// LS Electric XG5000 project: 66_3_A
// PLC NewPLC
// module base 0 slot 0: 입출력 모듈:XBC-DR20S (DC 24V 입력 12점, 릴레이 출력 8점)

PROGRAM NewProgram (task: 스캔 프로그램)

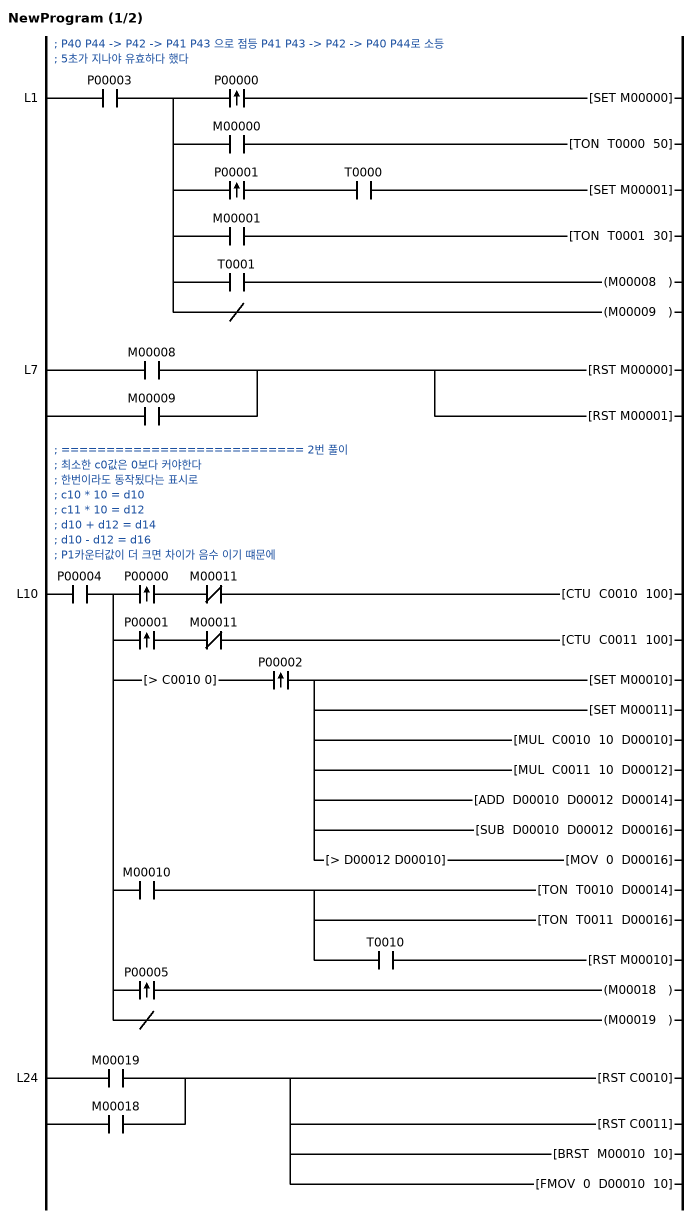
// P40 P44 -> P42 -> P41 P43 으로 점등 P41 P43 -> P42 -> P40 P44로 소등
; L1
LOAD      P00003
MPUSH
ANDP      P00000
SET       M00000
MLOAD
AND       M00000
TON       T0000 50
MLOAD
ANDP      P00001
AND       T0000
SET       M00001
MLOAD
AND       M00001
TON       T0001 30
MLOAD
AND       T0001
OUT       M00008
MPOP
NOT
OUT       M00009
// output comment: 5초가 지나야 유효하다 했다
; L7
LOAD      M00008
OR        M00009
RST       M00000
RST       M00001
// =========================== 2번 풀이
; L10
LOAD      P00004
MPUSH
ANDP      P00000
AND NOT   M00011
CTU       C0010 100
MLOAD
ANDP      P00001
AND NOT   M00011
CTU       C0011 100
MLOAD
AND>      C0010 0
ANDP      P00002
SET       M00010
SET       M00011
MUL       C0010 10 D00010
MUL       C0011 10 D00012
ADD       D00010 D00012 D00014
SUB       D00010 D00012 D00016
AND>      D00012 D00010
MOV       0 D00016
MLOAD
AND       M00010
TON       T0010 D00014
TON       T0011 D00016
AND       T0010
RST       M00010
MLOAD
ANDP      P00005
OUT       M00018
MPOP
NOT
OUT       M00019
// output comment: 
// output comment: 최소한 c0값은 0보다 커야한다
// output comment: 한번이라도 동작됬다는 표시로
// output comment: c10 * 10 = d10
// output comment: c11 * 10 = d12
// output comment: d10 + d12 = d14
// output comment: d10 - d12 = d16
// output comment: P1카운터값이 더 크면 차이가 음수 이기 떄문에
; L24
LOAD      M00019
OR        M00018
RST       C0010
RST       C0011
BRST      M00010 10
FMOV      0 D00010 10

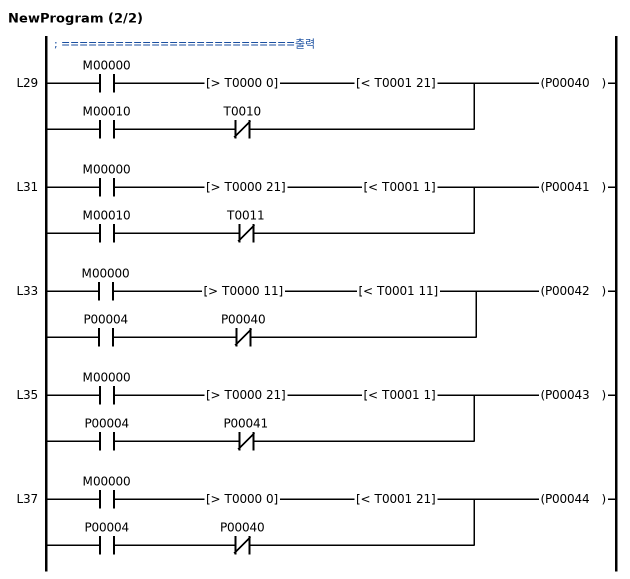
// ==========================출력
; L29
LOAD      M00000
AND>      T0000 0
AND<      T0001 21
LOAD      M00010
AND NOT   T0010
OR LOAD
OUT       P00040
; L31
LOAD      M00000
AND>      T0000 21
AND<      T0001 1
LOAD      M00010
AND NOT   T0011
OR LOAD
OUT       P00041
; L33
LOAD      M00000
AND>      T0000 11
AND<      T0001 11
LOAD      P00004
AND NOT   P00040
OR LOAD
OUT       P00042
; L35
LOAD      M00000
AND>      T0000 21
AND<      T0001 1
LOAD      P00004
AND NOT   P00041
OR LOAD
OUT       P00043
; L37
LOAD      M00000
AND>      T0000 0
AND<      T0001 21
LOAD      P00004
AND NOT   P00040
OR LOAD
OUT       P00044